Staubli VAL3: onLeftEvent.pgx

program onLeftEvent()
  local num i
  local num l_nDefault
begin
  // left click
  //
  // select the previous one
  //
  nProgID=(size(saveData:sProgType)+nProgID-1)%size(saveData:sProgType)
  if nProgID!=2
    sProgType=saveData:sProgType[nProgID]
  else
    // maintenance program
    sProgType=saveData:sProgType[0]
  endIf
  // load the progType
  call load()
  // rebuild the list
  call buildList()
  // refresh
  use:bUseRefresh=true
end
